// TIA Portal V17 export
// export: Created 2023-02-14T02:49:14.2245256Z, ExportSetting WithDefaults, DisplayName Totally Integrated Automation Portal, DisplayVersion V17, DisplayName TIA Portal Openness, DisplayVersion V17, DisplayName TIA Portal Teamcenter Gateway, DisplayVersion V17, DisplayName TIA Portal Version Control Interface, DisplayVersion V17, DisplayName SINAMICS Startdrive Advanced, DisplayVersion V17, DisplayName SINAMICS Startdrive G130, G150, S120, S150, SINAMICS MV, S210, DisplayVersion V17, DisplayName SINAMICS Startdrive G110M, G120, G120C, G120D, G120P, G115D, DisplayVersion V17, DisplayName STEP 7 Professional, DisplayVersion V17, DisplayName STEP 7 Safety, DisplayVersion V17, DisplayName WinCC Professional, DisplayVersion V17
DATA_BLOCK "Blend to Preparation"   // DB461
{ S7_Optimized_Access := 'TRUE' }
VERSION : 0.1
// stored: AutoNumber false, DBAccessibleFromOPCUA true, DBAccessibleFromWebserver true, IsOnlyStoredInLoadMemory false, IsRetainMemResEnabled false, IsWriteProtectedInAS false, MemoryReserve 0
   VAR
      "T-20" : Struct
         Raw_Material : Struct
            HW : Struct
               DoseRun : Bool;
               DoseHeld : Bool;
               DoseComplete : Bool;
               ValveCMD : Bool;
               PumpCMD : Bool;
               Header1_Req : Bool;
               Header2_Req : Bool;
            END_STRUCT;
            ChiliAwetan_1 : Struct
               DoseRun : Bool;
               DoseHeld : Bool;
               DoseComplete : Bool;
               ValveCMD : Bool;
               PumpCMD : Bool;
               Header1_Req : Bool;
               Header2_Req : Bool;
            END_STRUCT;
            ChiliAwetan_2 : Struct
               DoseRun : Bool;
               DoseHeld : Bool;
               DoseComplete : Bool;
               ValveCMD : Bool;
               PumpCMD : Bool;
               Header1_Req : Bool;
               Header2_Req : Bool;
            END_STRUCT;
            ChiliAwetan_3 : Struct
               DoseRun : Bool;
               DoseHeld : Bool;
               DoseComplete : Bool;
               ValveCMD : Bool;
               PumpCMD : Bool;
               Header1_Req : Bool;
               Header2_Req : Bool;
            END_STRUCT;
            Tomato : Struct
               DoseRun : Bool;
               DoseHeld : Bool;
               DoseComplete : Bool;
               ValveCMD : Bool;
               PumpCMD : Bool;
               Header1_Req : Bool;
               Header2_Req : Bool;
            END_STRUCT;
            ChiliFresh_1 : Struct
               DoseRun : Bool;
               DoseHeld : Bool;
               DoseComplete : Bool;
               ValveCMD : Bool;
               PumpCMD : Bool;
               Header1_Req : Bool;
               Header2_Req : Bool;
            END_STRUCT;
            ChiliFresh_2 : Struct
               DoseRun : Bool;
               DoseHeld : Bool;
               DoseComplete : Bool;
               ValveCMD : Bool;
               PumpCMD : Bool;
               Header1_Req : Bool;
               Header2_Req : Bool;
            END_STRUCT;
            ChiliFresh_3 : Struct
               DoseRun : Bool;
               DoseHeld : Bool;
               DoseComplete : Bool;
               ValveCMD : Bool;
               PumpCMD : Bool;
               Header1_Req : Bool;
               Header2_Req : Bool;
            END_STRUCT;
            Garlic : Struct
               DoseRun : Bool;
               DoseHeld : Bool;
               DoseComplete : Bool;
               ValveCMD : Bool;
               PumpCMD : Bool;
               Header1_Req : Bool;
               Header2_Req : Bool;
            END_STRUCT;
            Vinegar : Struct
               DoseRun : Bool;
               DoseHeld : Bool;
               DoseComplete : Bool;
               ValveCMD : Bool;
               PumpCMD : Bool;
               Header1_Req : Bool;
               Header2_Req : Bool;
            END_STRUCT;
         END_STRUCT;
         LineHeader1_OK : Bool;
         LineHeader2_OK : Bool;
         LineVinegar_OK : Bool;
         freeBool_4 : Bool;
         freeBool_5 : Bool;
         freeReal_1 : Bool;
         freeReal_2 : Bool;
         freeReal_3 : Bool;
         freeReal_4 : Bool;
         freeReal_5 : Bool;
      END_STRUCT;
      "T-21" : Struct
         Raw_Material : Struct
            HW : Struct
               DoseRun : Bool;
               DoseHeld : Bool;
               DoseComplete : Bool;
               ValveCMD : Bool;
               PumpCMD : Bool;
               Header1_Req : Bool;
               Header2_Req : Bool;
            END_STRUCT;
            ChiliAwetan_1 : Struct
               DoseRun : Bool;
               DoseHeld : Bool;
               DoseComplete : Bool;
               ValveCMD : Bool;
               PumpCMD : Bool;
               Header1_Req : Bool;
               Header2_Req : Bool;
            END_STRUCT;
            ChiliAwetan_2 : Struct
               DoseRun : Bool;
               DoseHeld : Bool;
               DoseComplete : Bool;
               ValveCMD : Bool;
               PumpCMD : Bool;
               Header1_Req : Bool;
               Header2_Req : Bool;
            END_STRUCT;
            ChiliAwetan_3 : Struct
               DoseRun : Bool;
               DoseHeld : Bool;
               DoseComplete : Bool;
               ValveCMD : Bool;
               PumpCMD : Bool;
               Header1_Req : Bool;
               Header2_Req : Bool;
            END_STRUCT;
            Tomato : Struct
               DoseRun : Bool;
               DoseHeld : Bool;
               DoseComplete : Bool;
               ValveCMD : Bool;
               PumpCMD : Bool;
               Header1_Req : Bool;
               Header2_Req : Bool;
            END_STRUCT;
            ChiliFresh_1 : Struct
               DoseRun : Bool;
               DoseHeld : Bool;
               DoseComplete : Bool;
               ValveCMD : Bool;
               PumpCMD : Bool;
               Header1_Req : Bool;
               Header2_Req : Bool;
            END_STRUCT;
            ChiliFresh_2 : Struct
               DoseRun : Bool;
               DoseHeld : Bool;
               DoseComplete : Bool;
               ValveCMD : Bool;
               PumpCMD : Bool;
               Header1_Req : Bool;
               Header2_Req : Bool;
            END_STRUCT;
            ChiliFresh_3 : Struct
               DoseRun : Bool;
               DoseHeld : Bool;
               DoseComplete : Bool;
               ValveCMD : Bool;
               PumpCMD : Bool;
               Header1_Req : Bool;
               Header2_Req : Bool;
            END_STRUCT;
            Garlic : Struct
               DoseRun : Bool;
               DoseHeld : Bool;
               DoseComplete : Bool;
               ValveCMD : Bool;
               PumpCMD : Bool;
               Header1_Req : Bool;
               Header2_Req : Bool;
            END_STRUCT;
            Vinegar : Struct
               DoseRun : Bool;
               DoseHeld : Bool;
               DoseComplete : Bool;
               ValveCMD : Bool;
               PumpCMD : Bool;
               Header1_Req : Bool;
               Header2_Req : Bool;
            END_STRUCT;
         END_STRUCT;
         LineHeader1_OK : Bool;
         LineHeader2_OK : Bool;
         LineVinegar_OK : Bool;
         freeBool_4 : Bool;
         freeBool_5 : Bool;
         freeReal_1 : Bool;
         freeReal_2 : Bool;
         freeReal_3 : Bool;
         freeReal_4 : Bool;
         freeReal_5 : Bool;
      END_STRUCT;
      "T-30" : Struct
         Raw_Material : Struct
            HW : Struct
               DoseRun : Bool;
               DoseHeld : Bool;
               DoseComplete : Bool;
               ValveCMD : Bool;
               PumpCMD : Bool;
               Header1_Req : Bool;
               Header2_Req : Bool;
            END_STRUCT;
            ChiliAwetan_1 : Struct
               DoseRun : Bool;
               DoseHeld : Bool;
               DoseComplete : Bool;
               ValveCMD : Bool;
               PumpCMD : Bool;
               Header1_Req : Bool;
               Header2_Req : Bool;
            END_STRUCT;
            ChiliAwetan_2 : Struct
               DoseRun : Bool;
               DoseHeld : Bool;
               DoseComplete : Bool;
               ValveCMD : Bool;
               PumpCMD : Bool;
               Header1_Req : Bool;
               Header2_Req : Bool;
            END_STRUCT;
            ChiliAwetan_3 : Struct
               DoseRun : Bool;
               DoseHeld : Bool;
               DoseComplete : Bool;
               ValveCMD : Bool;
               PumpCMD : Bool;
               Header1_Req : Bool;
               Header2_Req : Bool;
            END_STRUCT;
            Tomato : Struct
               DoseRun : Bool;
               DoseHeld : Bool;
               DoseComplete : Bool;
               ValveCMD : Bool;
               PumpCMD : Bool;
               Header1_Req : Bool;
               Header2_Req : Bool;
            END_STRUCT;
            ChiliFresh_1 : Struct
               DoseRun : Bool;
               DoseHeld : Bool;
               DoseComplete : Bool;
               ValveCMD : Bool;
               PumpCMD : Bool;
               Header1_Req : Bool;
               Header2_Req : Bool;
            END_STRUCT;
            ChiliFresh_2 : Struct
               DoseRun : Bool;
               DoseHeld : Bool;
               DoseComplete : Bool;
               ValveCMD : Bool;
               PumpCMD : Bool;
               Header1_Req : Bool;
               Header2_Req : Bool;
            END_STRUCT;
            ChiliFresh_3 : Struct
               DoseRun : Bool;
               DoseHeld : Bool;
               DoseComplete : Bool;
               ValveCMD : Bool;
               PumpCMD : Bool;
               Header1_Req : Bool;
               Header2_Req : Bool;
            END_STRUCT;
            Garlic : Struct
               DoseRun : Bool;
               DoseHeld : Bool;
               DoseComplete : Bool;
               ValveCMD : Bool;
               PumpCMD : Bool;
               Header1_Req : Bool;
               Header2_Req : Bool;
            END_STRUCT;
            Vinegar : Struct
               DoseRun : Bool;
               DoseHeld : Bool;
               DoseComplete : Bool;
               ValveCMD : Bool;
               PumpCMD : Bool;
               Header1_Req : Bool;
               Header2_Req : Bool;
            END_STRUCT;
         END_STRUCT;
         LineHeader1_OK : Bool;
         LineHeader2_OK : Bool;
         LineVinegar_OK : Bool;
         freeBool_4 : Bool;
         freeBool_5 : Bool;
         freeReal_1 : Bool;
         freeReal_2 : Bool;
         freeReal_3 : Bool;
         freeReal_4 : Bool;
         freeReal_5 : Bool;
      END_STRUCT;
      "T-31" : Struct
         Raw_Material : Struct
            HW : Struct
               DoseRun : Bool;
               DoseHeld : Bool;
               DoseComplete : Bool;
               ValveCMD : Bool;
               PumpCMD : Bool;
               Header1_Req : Bool;
               Header2_Req : Bool;
            END_STRUCT;
            ChiliAwetan_1 : Struct
               DoseRun : Bool;
               DoseHeld : Bool;
               DoseComplete : Bool;
               ValveCMD : Bool;
               PumpCMD : Bool;
               Header1_Req : Bool;
               Header2_Req : Bool;
            END_STRUCT;
            ChiliAwetan_2 : Struct
               DoseRun : Bool;
               DoseHeld : Bool;
               DoseComplete : Bool;
               ValveCMD : Bool;
               PumpCMD : Bool;
               Header1_Req : Bool;
               Header2_Req : Bool;
            END_STRUCT;
            ChiliAwetan_3 : Struct
               DoseRun : Bool;
               DoseHeld : Bool;
               DoseComplete : Bool;
               ValveCMD : Bool;
               PumpCMD : Bool;
               Header1_Req : Bool;
               Header2_Req : Bool;
            END_STRUCT;
            Tomato : Struct
               DoseRun : Bool;
               DoseHeld : Bool;
               DoseComplete : Bool;
               ValveCMD : Bool;
               PumpCMD : Bool;
               Header1_Req : Bool;
               Header2_Req : Bool;
            END_STRUCT;
            ChiliFresh_1 : Struct
               DoseRun : Bool;
               DoseHeld : Bool;
               DoseComplete : Bool;
               ValveCMD : Bool;
               PumpCMD : Bool;
               Header1_Req : Bool;
               Header2_Req : Bool;
            END_STRUCT;
            ChiliFresh_2 : Struct
               DoseRun : Bool;
               DoseHeld : Bool;
               DoseComplete : Bool;
               ValveCMD : Bool;
               PumpCMD : Bool;
               Header1_Req : Bool;
               Header2_Req : Bool;
            END_STRUCT;
            ChiliFresh_3 : Struct
               DoseRun : Bool;
               DoseHeld : Bool;
               DoseComplete : Bool;
               ValveCMD : Bool;
               PumpCMD : Bool;
               Header1_Req : Bool;
               Header2_Req : Bool;
            END_STRUCT;
            Garlic : Struct
               DoseRun : Bool;
               DoseHeld : Bool;
               DoseComplete : Bool;
               ValveCMD : Bool;
               PumpCMD : Bool;
               Header1_Req : Bool;
               Header2_Req : Bool;
            END_STRUCT;
            Vinegar : Struct
               DoseRun : Bool;
               DoseHeld : Bool;
               DoseComplete : Bool;
               ValveCMD : Bool;
               PumpCMD : Bool;
               Header1_Req : Bool;
               Header2_Req : Bool;
            END_STRUCT;
         END_STRUCT;
         LineHeader1_OK : Bool;
         LineHeader2_OK : Bool;
         LineVinegar_OK : Bool;
         freeBool_4 : Bool;
         freeBool_5 : Bool;
         freeReal_1 : Bool;
         freeReal_2 : Bool;
         freeReal_3 : Bool;
         freeReal_4 : Bool;
         freeReal_5 : Bool;
      END_STRUCT;
      "T-40" : Struct
         Raw_Material : Struct
            HW : Struct
               DoseRun : Bool;
               DoseHeld : Bool;
               DoseComplete : Bool;
               ValveCMD : Bool;
               PumpCMD : Bool;
               Header1_Req : Bool;
               Header2_Req : Bool;
            END_STRUCT;
            ChiliAwetan_1 : Struct
               DoseRun : Bool;
               DoseHeld : Bool;
               DoseComplete : Bool;
               ValveCMD : Bool;
               PumpCMD : Bool;
               Header1_Req : Bool;
               Header2_Req : Bool;
            END_STRUCT;
            ChiliAwetan_2 : Struct
               DoseRun : Bool;
               DoseHeld : Bool;
               DoseComplete : Bool;
               ValveCMD : Bool;
               PumpCMD : Bool;
               Header1_Req : Bool;
               Header2_Req : Bool;
            END_STRUCT;
            ChiliAwetan_3 : Struct
               DoseRun : Bool;
               DoseHeld : Bool;
               DoseComplete : Bool;
               ValveCMD : Bool;
               PumpCMD : Bool;
               Header1_Req : Bool;
               Header2_Req : Bool;
            END_STRUCT;
            Tomato : Struct
               DoseRun : Bool;
               DoseHeld : Bool;
               DoseComplete : Bool;
               ValveCMD : Bool;
               PumpCMD : Bool;
               Header1_Req : Bool;
               Header2_Req : Bool;
            END_STRUCT;
            ChiliFresh_1 : Struct
               DoseRun : Bool;
               DoseHeld : Bool;
               DoseComplete : Bool;
               ValveCMD : Bool;
               PumpCMD : Bool;
               Header1_Req : Bool;
               Header2_Req : Bool;
            END_STRUCT;
            ChiliFresh_2 : Struct
               DoseRun : Bool;
               DoseHeld : Bool;
               DoseComplete : Bool;
               ValveCMD : Bool;
               PumpCMD : Bool;
               Header1_Req : Bool;
               Header2_Req : Bool;
            END_STRUCT;
            ChiliFresh_3 : Struct
               DoseRun : Bool;
               DoseHeld : Bool;
               DoseComplete : Bool;
               ValveCMD : Bool;
               PumpCMD : Bool;
               Header1_Req : Bool;
               Header2_Req : Bool;
            END_STRUCT;
            Garlic : Struct
               DoseRun : Bool;
               DoseHeld : Bool;
               DoseComplete : Bool;
               ValveCMD : Bool;
               PumpCMD : Bool;
               Header1_Req : Bool;
               Header2_Req : Bool;
            END_STRUCT;
            Vinegar : Struct
               DoseRun : Bool;
               DoseHeld : Bool;
               DoseComplete : Bool;
               ValveCMD : Bool;
               PumpCMD : Bool;
               Header1_Req : Bool;
               Header2_Req : Bool;
            END_STRUCT;
         END_STRUCT;
         LineHeader1_OK : Bool;
         LineHeader2_OK : Bool;
         LineVinegar_OK : Bool;
         freeBool_4 : Bool;
         freeBool_5 : Bool;
         freeReal_1 : Bool;
         freeReal_2 : Bool;
         freeReal_3 : Bool;
         freeReal_4 : Bool;
         freeReal_5 : Bool;
      END_STRUCT;
      "T-41" : Struct
         Raw_Material : Struct
            HW : Struct
               DoseRun : Bool;
               DoseHeld : Bool;
               DoseComplete : Bool;
               ValveCMD : Bool;
               PumpCMD : Bool;
               Header1_Req : Bool;
               Header2_Req : Bool;
            END_STRUCT;
            ChiliAwetan_1 : Struct
               DoseRun : Bool;
               DoseHeld : Bool;
               DoseComplete : Bool;
               ValveCMD : Bool;
               PumpCMD : Bool;
               Header1_Req : Bool;
               Header2_Req : Bool;
            END_STRUCT;
            ChiliAwetan_2 : Struct
               DoseRun : Bool;
               DoseHeld : Bool;
               DoseComplete : Bool;
               ValveCMD : Bool;
               PumpCMD : Bool;
               Header1_Req : Bool;
               Header2_Req : Bool;
            END_STRUCT;
            ChiliAwetan_3 : Struct
               DoseRun : Bool;
               DoseHeld : Bool;
               DoseComplete : Bool;
               ValveCMD : Bool;
               PumpCMD : Bool;
               Header1_Req : Bool;
               Header2_Req : Bool;
            END_STRUCT;
            Tomato : Struct
               DoseRun : Bool;
               DoseHeld : Bool;
               DoseComplete : Bool;
               ValveCMD : Bool;
               PumpCMD : Bool;
               Header1_Req : Bool;
               Header2_Req : Bool;
            END_STRUCT;
            ChiliFresh_1 : Struct
               DoseRun : Bool;
               DoseHeld : Bool;
               DoseComplete : Bool;
               ValveCMD : Bool;
               PumpCMD : Bool;
               Header1_Req : Bool;
               Header2_Req : Bool;
            END_STRUCT;
            ChiliFresh_2 : Struct
               DoseRun : Bool;
               DoseHeld : Bool;
               DoseComplete : Bool;
               ValveCMD : Bool;
               PumpCMD : Bool;
               Header1_Req : Bool;
               Header2_Req : Bool;
            END_STRUCT;
            ChiliFresh_3 : Struct
               DoseRun : Bool;
               DoseHeld : Bool;
               DoseComplete : Bool;
               ValveCMD : Bool;
               PumpCMD : Bool;
               Header1_Req : Bool;
               Header2_Req : Bool;
            END_STRUCT;
            Garlic : Struct
               DoseRun : Bool;
               DoseHeld : Bool;
               DoseComplete : Bool;
               ValveCMD : Bool;
               PumpCMD : Bool;
               Header1_Req : Bool;
               Header2_Req : Bool;
            END_STRUCT;
            Vinegar : Struct
               DoseRun : Bool;
               DoseHeld : Bool;
               DoseComplete : Bool;
               ValveCMD : Bool;
               PumpCMD : Bool;
               Header1_Req : Bool;
               Header2_Req : Bool;
            END_STRUCT;
         END_STRUCT;
         LineHeader1_OK : Bool;
         LineHeader2_OK : Bool;
         LineVinegar_OK : Bool;
         freeBool_4 : Bool;
         freeBool_5 : Bool;
         freeReal_1 : Bool;
         freeReal_2 : Bool;
         freeReal_3 : Bool;
         freeReal_4 : Bool;
         freeReal_5 : Bool;
      END_STRUCT;
   END_VAR
   VAR RETAIN
      Recipe : Struct
         "T-20" : Struct
            HW : Struct
               Sp_Flush_to_BlendQty : Real;
               Sp_Flush_to_DrainQty : Real;
               Sp_DrainTime : DInt;
               SP_PumpSpeed : Real;
            END_STRUCT;
            ChiliAwetan_1 : Struct
               Sp_DoseQty : Real;
               SP_PumpSpeed : Real;
            END_STRUCT;
            ChiliAwetan_2 : Struct
               Sp_DoseQty : Real;
               SP_PumpSpeed : Real;
            END_STRUCT;
            ChiliAwetan_3 : Struct
               Sp_DoseQty : Real;
               SP_PumpSpeed : Real;
            END_STRUCT;
            Tomato : Struct
               Sp_DoseQty : Real;
               SP_PumpSpeed : Real;
            END_STRUCT;
            ChiliFresh_1 : Struct
               Sp_DoseQty : Real;
               SP_PumpSpeed : Real;
            END_STRUCT;
            ChiliFresh_2 : Struct
               Sp_DoseQty : Real;
               SP_PumpSpeed : Real;
            END_STRUCT;
            ChiliFresh_3 : Struct
               Sp_DoseQty : Real;
               SP_PumpSpeed : Real;
            END_STRUCT;
            Garlic : Struct
               Sp_DoseQty : Real;
               SP_PumpSpeed : Real;
            END_STRUCT;
            Vinegar : Struct
               Sp_DoseQty : Real;
               SP_PumpSpeed : Real;
            END_STRUCT;
            Sugar : Struct
               Sp_DoseQty : Real;
               SP_PumpSpeed : Real;
            END_STRUCT;
            Salt : Struct
               Sp_DoseQty : Real;
               SP_PumpSpeed : Real;
            END_STRUCT;
            ProWater : Struct
               Sp_DoseQty : Real;
               SP_PumpSpeed : Real;
            END_STRUCT;
            Homomixer : Struct
               Sp_DoseQty : Real;
               SP_PumpSpeed : Real;
            END_STRUCT;
         END_STRUCT;
         "T-21" : Struct
            HW : Struct
               Sp_Flush_to_BlendQty : Real;
               Sp_Flush_to_DrainQty : Real;
               Sp_DrainTime : DInt;
               SP_PumpSpeed : Real;
            END_STRUCT;
            ChiliAwetan_1 : Struct
               Sp_DoseQty : Real;
               SP_PumpSpeed : Real;
            END_STRUCT;
            ChiliAwetan_2 : Struct
               Sp_DoseQty : Real;
               SP_PumpSpeed : Real;
            END_STRUCT;
            ChiliAwetan_3 : Struct
               Sp_DoseQty : Real;
               SP_PumpSpeed : Real;
            END_STRUCT;
            Tomato : Struct
               Sp_DoseQty : Real;
               SP_PumpSpeed : Real;
            END_STRUCT;
            ChiliFresh_1 : Struct
               Sp_DoseQty : Real;
               SP_PumpSpeed : Real;
            END_STRUCT;
            ChiliFresh_2 : Struct
               Sp_DoseQty : Real;
               SP_PumpSpeed : Real;
            END_STRUCT;
            ChiliFresh_3 : Struct
               Sp_DoseQty : Real;
               SP_PumpSpeed : Real;
            END_STRUCT;
            Garlic : Struct
               Sp_DoseQty : Real;
               SP_PumpSpeed : Real;
            END_STRUCT;
            Vinegar : Struct
               Sp_DoseQty : Real;
               SP_PumpSpeed : Real;
            END_STRUCT;
            Sugar : Struct
               Sp_DoseQty : Real;
               SP_PumpSpeed : Real;
            END_STRUCT;
            Salt : Struct
               Sp_DoseQty : Real;
               SP_PumpSpeed : Real;
            END_STRUCT;
            ProWater : Struct
               Sp_DoseQty : Real;
               SP_PumpSpeed : Real;
            END_STRUCT;
            Homomixer : Struct
               Sp_DoseQty : Real;
               SP_PumpSpeed : Real;
            END_STRUCT;
         END_STRUCT;
         "T-30" : Struct
            HW : Struct
               Sp_Flush_to_BlendQty : Real;
               Sp_Flush_to_DrainQty : Real;
               Sp_DrainTime : DInt;
               SP_PumpSpeed : Real;
            END_STRUCT;
            ChiliAwetan_1 : Struct
               Sp_DoseQty : Real;
               SP_PumpSpeed : Real;
            END_STRUCT;
            ChiliAwetan_2 : Struct
               Sp_DoseQty : Real;
               SP_PumpSpeed : Real;
            END_STRUCT;
            ChiliAwetan_3 : Struct
               Sp_DoseQty : Real;
               SP_PumpSpeed : Real;
            END_STRUCT;
            Tomato : Struct
               Sp_DoseQty : Real;
               SP_PumpSpeed : Real;
            END_STRUCT;
            ChiliFresh_1 : Struct
               Sp_DoseQty : Real;
               SP_PumpSpeed : Real;
            END_STRUCT;
            ChiliFresh_2 : Struct
               Sp_DoseQty : Real;
               SP_PumpSpeed : Real;
            END_STRUCT;
            ChiliFresh_3 : Struct
               Sp_DoseQty : Real;
               SP_PumpSpeed : Real;
            END_STRUCT;
            Garlic : Struct
               Sp_DoseQty : Real;
               SP_PumpSpeed : Real;
            END_STRUCT;
            Vinegar : Struct
               Sp_DoseQty : Real;
               SP_PumpSpeed : Real;
            END_STRUCT;
            Sugar : Struct
               Sp_DoseQty : Real;
               SP_PumpSpeed : Real;
            END_STRUCT;
            Salt : Struct
               Sp_DoseQty : Real;
               SP_PumpSpeed : Real;
            END_STRUCT;
            ProWater : Struct
               Sp_DoseQty : Real;
               SP_PumpSpeed : Real;
            END_STRUCT;
            Homomixer : Struct
               Sp_DoseQty : Real;
               SP_PumpSpeed : Real;
            END_STRUCT;
         END_STRUCT;
         "T-31" : Struct
            HW : Struct
               Sp_Flush_to_BlendQty : Real;
               Sp_Flush_to_DrainQty : Real;
               Sp_DrainTime : DInt;
               SP_PumpSpeed : Real;
            END_STRUCT;
            ChiliAwetan_1 : Struct
               Sp_DoseQty : Real;
               SP_PumpSpeed : Real;
            END_STRUCT;
            ChiliAwetan_2 : Struct
               Sp_DoseQty : Real;
               SP_PumpSpeed : Real;
            END_STRUCT;
            ChiliAwetan_3 : Struct
               Sp_DoseQty : Real;
               SP_PumpSpeed : Real;
            END_STRUCT;
            Tomato : Struct
               Sp_DoseQty : Real;
               SP_PumpSpeed : Real;
            END_STRUCT;
            ChiliFresh_1 : Struct
               Sp_DoseQty : Real;
               SP_PumpSpeed : Real;
            END_STRUCT;
            ChiliFresh_2 : Struct
               Sp_DoseQty : Real;
               SP_PumpSpeed : Real;
            END_STRUCT;
            ChiliFresh_3 : Struct
               Sp_DoseQty : Real;
               SP_PumpSpeed : Real;
            END_STRUCT;
            Garlic : Struct
               Sp_DoseQty : Real;
               SP_PumpSpeed : Real;
            END_STRUCT;
            Vinegar : Struct
               Sp_DoseQty : Real;
               SP_PumpSpeed : Real;
            END_STRUCT;
            Sugar : Struct
               Sp_DoseQty : Real;
               SP_PumpSpeed : Real;
            END_STRUCT;
            Salt : Struct
               Sp_DoseQty : Real;
               SP_PumpSpeed : Real;
            END_STRUCT;
            ProWater : Struct
               Sp_DoseQty : Real;
               SP_PumpSpeed : Real;
            END_STRUCT;
            Homomixer : Struct
               Sp_DoseQty : Real;
               SP_PumpSpeed : Real;
            END_STRUCT;
         END_STRUCT;
         "T-40" : Struct
            HW : Struct
               Sp_Flush_to_BlendQty : Real;
               Sp_Flush_to_DrainQty : Real;
               Sp_DrainTime : DInt;
               SP_PumpSpeed : Real;
            END_STRUCT;
            ChiliAwetan_1 : Struct
               Sp_DoseQty : Real;
               SP_PumpSpeed : Real;
            END_STRUCT;
            ChiliAwetan_2 : Struct
               Sp_DoseQty : Real;
               SP_PumpSpeed : Real;
            END_STRUCT;
            ChiliAwetan_3 : Struct
               Sp_DoseQty : Real;
               SP_PumpSpeed : Real;
            END_STRUCT;
            Tomato : Struct
               Sp_DoseQty : Real;
               SP_PumpSpeed : Real;
            END_STRUCT;
            ChiliFresh_1 : Struct
               Sp_DoseQty : Real;
               SP_PumpSpeed : Real;
            END_STRUCT;
            ChiliFresh_2 : Struct
               Sp_DoseQty : Real;
               SP_PumpSpeed : Real;
            END_STRUCT;
            ChiliFresh_3 : Struct
               Sp_DoseQty : Real;
               SP_PumpSpeed : Real;
            END_STRUCT;
            Garlic : Struct
               Sp_DoseQty : Real;
               SP_PumpSpeed : Real;
            END_STRUCT;
            Vinegar : Struct
               Sp_DoseQty : Real;
               SP_PumpSpeed : Real;
            END_STRUCT;
            Sugar : Struct
               Sp_DoseQty : Real;
               SP_PumpSpeed : Real;
            END_STRUCT;
            Salt : Struct
               Sp_DoseQty : Real;
               SP_PumpSpeed : Real;
            END_STRUCT;
            ProWater : Struct
               Sp_DoseQty : Real;
               SP_PumpSpeed : Real;
            END_STRUCT;
            Homomixer : Struct
               Sp_DoseQty : Real;
               SP_PumpSpeed : Real;
            END_STRUCT;
         END_STRUCT;
         "T-41" : Struct
            HW : Struct
               Sp_Flush_to_BlendQty : Real;
               Sp_Flush_to_DrainQty : Real;
               Sp_DrainTime : DInt;
               SP_PumpSpeed : Real;
            END_STRUCT;
            ChiliAwetan_1 : Struct
               Sp_DoseQty : Real;
               SP_PumpSpeed : Real;
            END_STRUCT;
            ChiliAwetan_2 : Struct
               Sp_DoseQty : Real;
               SP_PumpSpeed : Real;
            END_STRUCT;
            ChiliAwetan_3 : Struct
               Sp_DoseQty : Real;
               SP_PumpSpeed : Real;
            END_STRUCT;
            Tomato : Struct
               Sp_DoseQty : Real;
               SP_PumpSpeed : Real;
            END_STRUCT;
            ChiliFresh_1 : Struct
               Sp_DoseQty : Real;
               SP_PumpSpeed : Real;
            END_STRUCT;
            ChiliFresh_2 : Struct
               Sp_DoseQty : Real;
               SP_PumpSpeed : Real;
            END_STRUCT;
            ChiliFresh_3 : Struct
               Sp_DoseQty : Real;
               SP_PumpSpeed : Real;
            END_STRUCT;
            Garlic : Struct
               Sp_DoseQty : Real;
               SP_PumpSpeed : Real;
            END_STRUCT;
            Vinegar : Struct
               Sp_DoseQty : Real;
               SP_PumpSpeed : Real;
            END_STRUCT;
            Sugar : Struct
               Sp_DoseQty : Real;
               SP_PumpSpeed : Real;
            END_STRUCT;
            Salt : Struct
               Sp_DoseQty : Real;
               SP_PumpSpeed : Real;
            END_STRUCT;
            ProWater : Struct
               Sp_DoseQty : Real;
               SP_PumpSpeed : Real;
            END_STRUCT;
            Homomixer : Struct
               Sp_DoseQty : Real;
               SP_PumpSpeed : Real;
            END_STRUCT;
         END_STRUCT;
      END_STRUCT;
   END_VAR
   VAR
      ProdReq_Header_1 : Bool;
      ProdReq_Header_2 : Bool;
      freeBool_3 : Bool;
      freeBool_4 : Bool;
      freeBool_5 : Bool;
      freeBool_6 : Bool;
      freeBool_7 : Bool;
      freeBool_8 : Bool;
      freeBool_9 : Bool;
      freeBool_10 : Bool;
      freeBool_11 : Bool;
      freeBool_12 : Bool;
      freeBool_13 : Bool;
      freeBool_14 : Bool;
      freeBool_15 : Bool;
      freeBool_16 : Bool;
      freeReal_1 : Real;
      freeReal_2 : Real;
      freeReal_3 : Real;
      freeReal_4 : Real;
      freeReal_5 : Real;
      freeReal_6 : Real;
      freeReal_7 : Real;
      freeReal_8 : Real;
      freeReal_9 : Real;
      freeReal_10 : Real;
      freeReal_11 : Real;
      freeReal_12 : Real;
      freeReal_13 : Real;
      freeReal_14 : Real;
      freeReal_15 : Real;
      freeReal_16 : Real;
   END_VAR
BEGIN
END_DATA_BLOCK
